{attribute 'GeneratedUsingTerminal: EL1258-0000-0016'}
{attribute addProperty BoxType "EL1258-0000-0016"}
{attribute addProperty Description "EL1258 8Ch. Dig Input 24V with Multi-Time-Stamp"}
{attribute addProperty Physics "KK"}
{attribute addProperty Id "MTI_Inputs_10x_Channel_1AT %I*MTI_Inputs_10x_Channel_C3ED30FD56MTI_Inputs_10x_Channel_2AT %I*MTI_Inputs_10x_Channel_C3ED30FD56MTI_Inputs_10x_Channel_3AT %I*MTI_Inputs_10x_Channel_C3ED30FD56MTI_Inputs_10x_Channel_4AT %I*MTI_Inputs_10x_Channel_C3ED30FD56MTI_Inputs_10x_Channel_5AT %I*MTI_Inputs_10x_Channel_C3ED30FD56MTI_Inputs_10x_Channel_6AT %I*MTI_Inputs_10x_Channel_C3ED30FD56MTI_Inputs_10x_Channel_7AT %I*MTI_Inputs_10x_Channel_C3ED30FD56MTI_Inputs_10x_Channel_8AT %I*MTI_Inputs_10x_Channel_C3ED30FD56MTI_Outputs_Channel_1AT %Q*MTI_Outputs_Channel_0F1028A12MTI_Outputs_Channel_2AT %Q*MTI_Outputs_Channel_0F1028A12MTI_Outputs_Channel_3AT %Q*MTI_Outputs_Channel_0F1028A12MTI_Outputs_Channel_4AT %Q*MTI_Outputs_Channel_0F1028A12MTI_Outputs_Channel_5AT %Q*MTI_Outputs_Channel_0F1028A12MTI_Outputs_Channel_6AT %Q*MTI_Outputs_Channel_0F1028A12MTI_Outputs_Channel_7AT %Q*MTI_Outputs_Channel_0F1028A12MTI_Outputs_Channel_8AT %Q*MTI_Outputs_Channel_0F1028A12WcStateAT %I*WcState_9091E0EB2InfoDataAT %I*InfoData_BEF6B88E18"}
{attribute addProperty CRC "1933509618"}
{attribute addProperty Size "484"}
TYPE EL1258_733F03F2 EXTENDS EtcSlaveTerminalBase_947E5A46 :
STRUCT
	{attribute addProperty Name "MTI_Inputs_10x_Channel_1"}
	MTI_Inputs_10x_Channel_1 : MTI_Inputs_10x_Channel_C3ED30FD;
	{attribute addProperty Name "MTI_Inputs_10x_Channel_2"}
	MTI_Inputs_10x_Channel_2 : MTI_Inputs_10x_Channel_C3ED30FD;
	{attribute addProperty Name "MTI_Inputs_10x_Channel_3"}
	MTI_Inputs_10x_Channel_3 : MTI_Inputs_10x_Channel_C3ED30FD;
	{attribute addProperty Name "MTI_Inputs_10x_Channel_4"}
	MTI_Inputs_10x_Channel_4 : MTI_Inputs_10x_Channel_C3ED30FD;
	{attribute addProperty Name "MTI_Inputs_10x_Channel_5"}
	MTI_Inputs_10x_Channel_5 : MTI_Inputs_10x_Channel_C3ED30FD;
	{attribute addProperty Name "MTI_Inputs_10x_Channel_6"}
	MTI_Inputs_10x_Channel_6 : MTI_Inputs_10x_Channel_C3ED30FD;
	{attribute addProperty Name "MTI_Inputs_10x_Channel_7"}
	MTI_Inputs_10x_Channel_7 : MTI_Inputs_10x_Channel_C3ED30FD;
	{attribute addProperty Name "MTI_Inputs_10x_Channel_8"}
	MTI_Inputs_10x_Channel_8 : MTI_Inputs_10x_Channel_C3ED30FD;
	{attribute addProperty Name "MTI_Outputs_Channel_1"}
	MTI_Outputs_Channel_1 : MTI_Outputs_Channel_0F1028A1;
	{attribute addProperty Name "MTI_Outputs_Channel_2"}
	MTI_Outputs_Channel_2 : MTI_Outputs_Channel_0F1028A1;
	{attribute addProperty Name "MTI_Outputs_Channel_3"}
	MTI_Outputs_Channel_3 : MTI_Outputs_Channel_0F1028A1;
	{attribute addProperty Name "MTI_Outputs_Channel_4"}
	MTI_Outputs_Channel_4 : MTI_Outputs_Channel_0F1028A1;
	{attribute addProperty Name "MTI_Outputs_Channel_5"}
	MTI_Outputs_Channel_5 : MTI_Outputs_Channel_0F1028A1;
	{attribute addProperty Name "MTI_Outputs_Channel_6"}
	MTI_Outputs_Channel_6 : MTI_Outputs_Channel_0F1028A1;
	{attribute addProperty Name "MTI_Outputs_Channel_7"}
	MTI_Outputs_Channel_7 : MTI_Outputs_Channel_0F1028A1;
	{attribute addProperty Name "MTI_Outputs_Channel_8"}
	MTI_Outputs_Channel_8 : MTI_Outputs_Channel_0F1028A1;
	{attribute addProperty Name "WcState"}
	WcState : WcState_9091E0EB;
	{attribute addProperty Name "InfoData"}
	InfoData : InfoData_BEF6B88E;
END_STRUCT
END_TYPE

(* stored: Version 1.2.0.0, ProductVersion 3.1.4024.11
   DUT EL1258_733F03F2: Id {0b54ff68-55c9-4d89-bf14-aa3e9a505ed5} *)
